// TIA Portal V18 export
TYPE "UDT_andonIO"
// stored: IsFailsafeCompliant false
   STRUCT
      I_greenBtn { ExternalVisible := 'False'; ExternalWritable := 'False'} : Bool;
      I_yellowBtn { ExternalVisible := 'False'; ExternalWritable := 'False'} : Bool;
      I_redBtn { ExternalVisible := 'False'; ExternalWritable := 'False'} : Bool;
      O_greenBtnLed { ExternalVisible := 'False'; ExternalWritable := 'False'} : Bool;
      O_yellowBtnLed { ExternalVisible := 'False'; ExternalWritable := 'False'} : Bool;
      O_redBtnLed { ExternalVisible := 'False'; ExternalWritable := 'False'} : Bool;
   END_STRUCT;
END_TYPE
